   ;FOLD SPTP P710 CONT Vel=100 % PDAT71 Tool[1] Base[0] ;%{PE}
      ;FOLD Parameters ;%{h}
         ;Params IlfProvider=kukaroboter.basistech.inlineforms.movement.spline; Kuka.IsGlobalPoint=FALSE; Kuka.PointName=P710; Kuka.BlendingEnabled=TRUE; Kuka.MoveDataPtpName=PDAT71; Kuka.VelocityPtp=100; Kuka.VelocityFieldEnabled=TRUE; Kuka.ColDetectFieldEnabled=TRUE; Kuka.CurrentCDSetIndex=0; Kuka.MovementParameterFieldEnabled=TRUE; IlfCommand=SPTP
      ;ENDFOLD
      SPTP XP710 WITH $VEL_AXIS[1] = SVEL_JOINT(100.0), $TOOL = STOOL2(FP710), $BASE = SBASE(FP710.BASE_NO), $IPO_MODE = SIPO_MODE(FP710.IPO_FRAME), $LOAD = SLOAD(FP710.TOOL_NO), $ACC_AXIS[1] = SACC_JOINT(PPDAT71), $APO = SAPO_PTP(PPDAT71), $GEAR_JERK[1] = SGEAR_JERK(PPDAT71), $COLLMON_TOL_PRO[1] = USE_CM_PRO_VALUES(0) C_Spl
   ;ENDFOLD

   trigger when distance=0 delay=0 do B_Brenner_aktiv=FALSE
   trigger when distance=1 delay=0 do Brenner (I_n_aktive_Brenner,#loeschen) prio=-1
   ;FOLD SPTP P700 CONT Vel=100 % PDAT72 Tool[1] Base[0] ;%{PE}
      ;FOLD Parameters ;%{h}
         ;Params IlfProvider=kukaroboter.basistech.inlineforms.movement.spline; Kuka.IsGlobalPoint=FALSE; Kuka.PointName=P700; Kuka.BlendingEnabled=TRUE; Kuka.MoveDataPtpName=PDAT72; Kuka.VelocityPtp=100; Kuka.VelocityFieldEnabled=TRUE; Kuka.ColDetectFieldEnabled=TRUE; Kuka.CurrentCDSetIndex=0; Kuka.MovementParameterFieldEnabled=TRUE; IlfCommand=SPTP
      ;ENDFOLD
      SPTP XP700 WITH $VEL_AXIS[1] = SVEL_JOINT(100.0), $TOOL = STOOL2(FP700), $BASE = SBASE(FP700.BASE_NO), $IPO_MODE = SIPO_MODE(FP700.IPO_FRAME), $LOAD = SLOAD(FP700.TOOL_NO), $ACC_AXIS[1] = SACC_JOINT(PPDAT72), $APO = SAPO_PTP(PPDAT72), $GEAR_JERK[1] = SGEAR_JERK(PPDAT72), $COLLMON_TOL_PRO[1] = USE_CM_PRO_VALUES(0) C_Spl
   ;ENDFOLD

END

;***************************************************
;** Alternativprogramm ohne Bauteilbeflammen *******
;***************************************************

DEF ohne_Beflammen ()

   ;BEFLAMMEN WIRD NICHT VERWENDET
   RETURN

   ; hier Roboterbewegung

   trigger when distance=1 delay=0 do UmgreifStation_Pos (#auf) prio=-1
   ;FOLD SPTP P1000 CONT Vel=100 % PDAT73 Tool[1] Base[0] ;%{PE}
      ;FOLD Parameters ;%{h}
         ;Params IlfProvider=kukaroboter.basistech.inlineforms.movement.spline; Kuka.IsGlobalPoint=FALSE; Kuka.PointName=P1000; Kuka.BlendingEnabled=TRUE; Kuka.MoveDataPtpName=PDAT73; Kuka.VelocityPtp=100; Kuka.VelocityFieldEnabled=TRUE; Kuka.ColDetectFieldEnabled=TRUE; Kuka.CurrentCDSetIndex=0; Kuka.MovementParameterFieldEnabled=TRUE; IlfCommand=SPTP
      ;ENDFOLD
      SPTP XP1000 WITH $VEL_AXIS[1] = SVEL_JOINT(100.0), $TOOL = STOOL2(FP1000), $BASE = SBASE(FP1000.BASE_NO), $IPO_MODE = SIPO_MODE(FP1000.IPO_FRAME), $LOAD = SLOAD(FP1000.TOOL_NO), $ACC_AXIS[1] = SACC_JOINT(PPDAT73), $APO = SAPO_PTP(PPDAT73), $GEAR_JERK[1] = SGEAR_JERK(PPDAT73), $COLLMON_TOL_PRO[1] = USE_CM_PRO_VALUES(0) C_Spl
   ;ENDFOLD

   continue
   if ((E_mit_Bedrucken==TRUE) and (B_Ausschuss==FALSE)) then ; $IN[1201] mit Bedrucken von SPS
      trigger when distance=1 delay=0 do drucker(#druck)prio=-1

   endif ; and (E_WAAGE_TEIL_IO)

   ;FOLD SPTP P1010 CONT Vel=100 % PDAT74 Tool[1] Base[0] ;%{PE}
      ;FOLD Parameters ;%{h}
         ;Params IlfProvider=kukaroboter.basistech.inlineforms.movement.spline; Kuka.IsGlobalPoint=FALSE; Kuka.PointName=P1010; Kuka.BlendingEnabled=TRUE; Kuka.MoveDataPtpName=PDAT74; Kuka.VelocityPtp=100; Kuka.VelocityFieldEnabled=TRUE; Kuka.ColDetectFieldEnabled=TRUE; Kuka.CurrentCDSetIndex=0; Kuka.MovementParameterFieldEnabled=TRUE; IlfCommand=SPTP
      ;ENDFOLD
      SPTP XP1010 WITH $VEL_AXIS[1] = SVEL_JOINT(100.0), $TOOL = STOOL2(FP1010), $BASE = SBASE(FP1010.BASE_NO), $IPO_MODE = SIPO_MODE(FP1010.IPO_FRAME), $LOAD = SLOAD(FP1010.TOOL_NO), $ACC_AXIS[1] = SACC_JOINT(PPDAT74), $APO = SAPO_PTP(PPDAT74), $GEAR_JERK[1] = SGEAR_JERK(PPDAT74), $COLLMON_TOL_PRO[1] = USE_CM_PRO_VALUES(0) C_Spl
   ;ENDFOLD

   if ((E_mit_Bedrucken==TRUE) and (B_Ausschuss==FALSE)) then ; $IN[1201] mit Bedrucken von SPS
      ; and (E_WAAGE_TEIL_IO)

      ;FOLD SPTP P1020 CONT Vel=100 % PDAT75 Tool[1] Base[0] ;%{PE}
         ;FOLD Parameters ;%{h}
            ;Params IlfProvider=kukaroboter.basistech.inlineforms.movement.spline; Kuka.IsGlobalPoint=FALSE; Kuka.PointName=P1020; Kuka.BlendingEnabled=TRUE; Kuka.MoveDataPtpName=PDAT75; Kuka.VelocityPtp=100; Kuka.VelocityFieldEnabled=TRUE; Kuka.ColDetectFieldEnabled=TRUE; Kuka.CurrentCDSetIndex=0; Kuka.MovementParameterFieldEnabled=TRUE; IlfCommand=SPTP
         ;ENDFOLD
         SPTP XP1020 WITH $VEL_AXIS[1] = SVEL_JOINT(100.0), $TOOL = STOOL2(FP1020), $BASE = SBASE(FP1020.BASE_NO), $IPO_MODE = SIPO_MODE(FP1020.IPO_FRAME), $LOAD = SLOAD(FP1020.TOOL_NO), $ACC_AXIS[1] = SACC_JOINT(PPDAT75), $APO = SAPO_PTP(PPDAT75), $GEAR_JERK[1] = SGEAR_JERK(PPDAT75), $COLLMON_TOL_PRO[1] = USE_CM_PRO_VALUES(0) C_Spl
      ;ENDFOLD
   endif

end
;***************************************************
;** Alternativprogramm ohne Bauteil bedrucken ******
;***************************************************

DEF ohne_RFID()

   ;Umorientierung wenn ohne RFID produziert wird

   ;FOLD SPTP P2000 CONT Vel=100 % PDAT76 Tool[1] Base[0] ;%{PE}
      ;FOLD Parameters ;%{h}
         ;Params IlfProvider=kukaroboter.basistech.inlineforms.movement.spline; Kuka.IsGlobalPoint=FALSE; Kuka.PointName=P2000; Kuka.BlendingEnabled=TRUE; Kuka.MoveDataPtpName=PDAT76; Kuka.VelocityPtp=100; Kuka.VelocityFieldEnabled=TRUE; Kuka.ColDetectFieldEnabled=TRUE; Kuka.CurrentCDSetIndex=0; Kuka.MovementParameterFieldEnabled=TRUE; IlfCommand=SPTP
      ;ENDFOLD
      SPTP XP2000 WITH $VEL_AXIS[1] = SVEL_JOINT(100.0), $TOOL = STOOL2(FP2000), $BASE = SBASE(FP2000.BASE_NO), $IPO_MODE = SIPO_MODE(FP2000.IPO_FRAME), $LOAD = SLOAD(FP2000.TOOL_NO), $ACC_AXIS[1] = SACC_JOINT(PPDAT76), $APO = SAPO_PTP(PPDAT76), $GEAR_JERK[1] = SGEAR_JERK(PPDAT76), $COLLMON_TOL_PRO[1] = USE_CM_PRO_VALUES(0) C_Spl
   ;ENDFOLD

   ;FOLD SPTP P2010 CONT Vel=100 % PDAT77 Tool[1] Base[0] ;%{PE}
      ;FOLD Parameters ;%{h}
         ;Params IlfProvider=kukaroboter.basistech.inlineforms.movement.spline; Kuka.IsGlobalPoint=FALSE; Kuka.PointName=P2010; Kuka.BlendingEnabled=TRUE; Kuka.MoveDataPtpName=PDAT77; Kuka.VelocityPtp=100; Kuka.VelocityFieldEnabled=TRUE; Kuka.ColDetectFieldEnabled=TRUE; Kuka.CurrentCDSetIndex=0; Kuka.MovementParameterFieldEnabled=TRUE; IlfCommand=SPTP
      ;ENDFOLD
      SPTP XP2010 WITH $VEL_AXIS[1] = SVEL_JOINT(100.0), $TOOL = STOOL2(FP2010), $BASE = SBASE(FP2010.BASE_NO), $IPO_MODE = SIPO_MODE(FP2010.IPO_FRAME), $LOAD = SLOAD(FP2010.TOOL_NO), $ACC_AXIS[1] = SACC_JOINT(PPDAT77), $APO = SAPO_PTP(PPDAT77), $GEAR_JERK[1] = SGEAR_JERK(PPDAT77), $COLLMON_TOL_PRO[1] = USE_CM_PRO_VALUES(0) C_Spl
   ;ENDFOLD

   ;FOLD SPTP P2020 CONT Vel=100 % PDAT78 Tool[1] Base[0] ;%{PE}
      ;FOLD Parameters ;%{h}
         ;Params IlfProvider=kukaroboter.basistech.inlineforms.movement.spline; Kuka.IsGlobalPoint=FALSE; Kuka.PointName=P2020; Kuka.BlendingEnabled=TRUE; Kuka.MoveDataPtpName=PDAT78; Kuka.VelocityPtp=100; Kuka.VelocityFieldEnabled=TRUE; Kuka.ColDetectFieldEnabled=TRUE; Kuka.CurrentCDSetIndex=0; Kuka.MovementParameterFieldEnabled=TRUE; IlfCommand=SPTP
      ;ENDFOLD
      SPTP XP2020 WITH $VEL_AXIS[1] = SVEL_JOINT(100.0), $TOOL = STOOL2(FP2020), $BASE = SBASE(FP2020.BASE_NO), $IPO_MODE = SIPO_MODE(FP2020.IPO_FRAME), $LOAD = SLOAD(FP2020.TOOL_NO), $ACC_AXIS[1] = SACC_JOINT(PPDAT78), $APO = SAPO_PTP(PPDAT78), $GEAR_JERK[1] = SGEAR_JERK(PPDAT78), $COLLMON_TOL_PRO[1] = USE_CM_PRO_VALUES(0) C_Spl
   ;ENDFOLD

end

;***************************************************
;** Programm, um rueckwaerts aus der Form bis vor **
;***        Teileaufnahme zu fahren              ***
;***************************************************

DEF  RRaus ( )

   INT i

   B_Ausschuss=TRUE
   $ov_pro=10
   BAS (#vel_cp,1.0)
   BAS (#vel_ptp,50)

   ventile_aus ()

   $BASE=Base_Data[1]
   $TOOL=Tool_Data[1]

   wait for (E_SGM_Form_auf==TRUE) ; $IN[3] SGM Form offen (E67)
   if ($flag[7]==TRUE) then
      LIN  XP100
   endif

   if ($flag[6]==TRUE) then
      LIN  XP40
   endif

   if ($flag[5]==TRUE) then
      LIN  XP35
   endif

   if ($flag[4]==TRUE) then
      LIN  XP30
   endif

   if ($flag[3]==TRUE) then
      PTP XP20
   endif

   if ($flag[2]==TRUE) then
      PTP XP10
   endif

   if ($flag[1]==TRUE) then
      PTP XHome
   else
      Meldung (#notify,10)
      Meldung (#quit,27)
      loop
         HALT  ;Roboter von Hand aus der Form fahren !!!
      endloop
   endif

   for i=1 to 10
      $flag[i]=FALSE
   endfor

   B_GST_war_gedrueckt=FALSE
   ;B_L_Start=FALSE
   B_Teilaufnahme=TRUE

END

;***************************************************
;** Programm, zum Uberpruefen der Endlagen der   **
;***            Benutzerventile                  ***
;***************************************************

Def Chk_BV (BV_Nr: in,BV_Zustand: in)

   INT BV_Nr
   DECL Mode2 BV_Zustand

   ;fold  Greiferbelegung, Stand: 02.11.2020
      ;***************************************************
      ;  V1  = Teilevakuum vorne
      ;  V2  = n.v.
      ;  V3  = Teilevakuum vorne unten ;nur ab Umgreifstation
      ;  V4  = Teilevakuum hinten unten ;nur ab Umgreifstation
      ;  BV1/AS = Teilegreifer schließen
      ;  BV1/GS = n.v.
      ;  BV2/AS = Teilegreifer hinten langer hub nach vorne
      ;  BV2/GS = Teilegreifer hinten langer hub nach hinten
      ;  BV3/AS = Teilegreifer hinten kurzer hub nach vorne
      ;  BV3/GS = Teilegreifer hinten kurzer hub nach hinten
      ;  BV4/AS = Angussgreifer schließen
      ;  BV4/GS = n.v.
      ;  BV5/AS = Angussschneider nach vorne
      ;  BV5/GS = Angussschneider nach hinten
      ;  BV6/AS = Angussschneider schließen
      ;***************************************************
   ;endfold

   switch BV_Nr

      ; Benutzerventil 1 = Teilegreifer
      case 1

         switch BV_Zustand

            case #GS

            case #AS

               wait for (E_ASi_22_3==TRUE); IN 363(Abf. Radl oben links)
               wait for (E_ASi_22_4==TRUE); IN 364(Abf. Dreilaendereck links)
               wait for (E_ASi_24_3==TRUE); IN 379(Abf. Radl unten links)
               wait for (E_ASi_26_3==TRUE); IN 395(Abf. Radl oben rechts)
               wait for (E_ASi_26_4==TRUE); IN 496(Abf. Dreilaendereck rechts)
               wait for (E_ASi_28_3==TRUE); IN 411(Abf. Radlauf unten rechts)

         endswitch

         ; Benutzerventil 2 =  Teilegreifer hinten langer hub
      case 2

         switch BV_Zustand

            case #GS

               wait for (E_ASi_22_1==TRUE)
               wait for (E_ASi_24_1==TRUE)
               wait for (E_ASi_26_1==TRUE)
               wait for (E_ASi_28_1==TRUE)

            case #AS

               wait for (E_ASi_22_2==TRUE)
               wait for (E_ASi_24_2==TRUE)
               wait for (E_ASi_26_2==TRUE)
               wait for (E_ASi_28_2==TRUE)

         endswitch

         ; Benutzerventil 3 = none
      case 3

         switch BV_Zustand

            case #GS

            case #AS

         endswitch

         ; Benutzerventil 4 = Angussgreifer
      case 4

         switch BV_Zustand

            case #GS

            case #AS

               wait for (E_ASi_23_1==TRUE); IN 369(Anguss links)
               wait for (E_ASi_23_2==TRUE); IN 370(Anguss rechts)
               wait for (E_ASi_27_1==TRUE); IN 401(Anguss rechts)

         endswitch

         ; Benutzerventil 5 = none
      case 5

         switch BV_Zustand

            case #GS

            case #AS

         endswitch

         ; Benutzerventil 6 = none
      case 6

         switch BV_Zustand

            case #GS

            case #AS

         endswitch

      default
         loop
            halt ; BV nicht vorhanden
         endloop

   endswitch

end

;***************************************************
;*** Teileabfrage Vakuumkreise und ASI Eingänge  ***
;***************************************************

DEF Teileabfrage()

   wait for (E_VK1==TRUE)
   ;wait for (E_VK2==TRUE)
   ;wait for (E_VK3==TRUE)
   ;wait for (E_VK4==TRUE)
   wait for (E_ASi_22_3==TRUE); IN 363(Abf. Radl oben links)
   wait for (E_ASi_22_4==TRUE); IN 364(Abf. Dreilaendereck links)
   wait for (E_ASi_23_1==TRUE); IN 369(Anguss links)
   wait for (E_ASi_23_2==TRUE); IN 370(Anguss rechts)
   wait for (E_ASi_24_3==TRUE); IN 379(Abf. Radl unten links)
   wait for (E_ASi_26_3==TRUE); IN 395(Abf. Radl oben rechts)
   wait for (E_ASi_26_4==TRUE); IN 496(Abf. Dreilaendereck rechts)
   wait for (E_ASi_27_1==TRUE); IN 401(Anguss rechts)
   wait for (E_ASi_28_3==TRUE); IN 411(Abf. Radlauf unten rechts)

End

--- sp15_005.dat ---
&ACCESS RVO1
&REL 244
&PARAM DISKPATH = KRC:\R1\Program\Bauteilprogramme
DEFDAT  SP15_005
;FOLD EXTERNAL DECLARATIONS;%{PE}%MKUKATPBASIS,%CEXT,%VCOMMON,%P
;FOLD BASISTECH EXT;%{PE}%MKUKATPBASIS,%CEXT,%VEXT,%P
EXT  BAS (BAS_COMMAND  :IN,REAL  :IN )
;ENDFOLD (BASISTECH EXT)
;FOLD USER EXT;%{E}%MKUKATPUSER,%CEXT,%VEXT,%P
;Make your modifications here

;ENDFOLD (USER EXT)
;ENDFOLD (EXTERNAL DECLARATIONS)

;***************************************************
;Common Declarations********************************
;***************************************************
DECL E6POS XP200={X 2198.25366,Y -125.542969,Z 1747.09790,A 176.729721,B 44.9991875,C 179.999023,S 2,T 34,E1 0.0,E2 0.0,E3 0.0,E4 0.0,E5 0.0,E6 0.0}
DECL FDAT FP200={TOOL_NO 1,BASE_NO 0,IPO_FRAME #BASE,POINT2[] " "}
DECL PDAT PPDAT6={VEL 100.000,ACC 100.000,APO_DIST 500.000,APO_MODE #CDIS,GEAR_JERK 100.000,EXAX_IGN 0}


;***************************************************
;SGM Declarations***********************************
;***************************************************
DECL E6POS XP10={X 1853.22363,Y 1615.74561,Z 1754.75720,A 60.7845039,B -43.4993439,C -175.197784,S 2,T 43,E1 0.0,E2 0.0,E3 0.0,E4 0.0,E5 0.0,E6 0.0}
DECL FDAT FP10={TOOL_NO 1,BASE_NO 0,IPO_FRAME #BASE,POINT2[] " "}
DECL PDAT PPDAT1={VEL 100.000,ACC 100.000,APO_DIST 250.000,APO_MODE #CDIS,GEAR_JERK 100.000,EXAX_IGN 0}

DECL E6POS XP20={X 1174.55273,Y 2717.27319,Z 949.700256,A -0.590916,B 44.9981651,C 179.820206,S 2,T 43,E1 0.0,E2 0.0,E3 0.0,E4 0.0,E5 0.0,E6 0.0}
DECL FDAT FP20={TOOL_NO 1,BASE_NO 0,IPO_FRAME #BASE,POINT2[] " "}
DECL PDAT PPDAT2={VEL 100.000,ACC 100.000,APO_DIST 250.000,APO_MODE #CDIS,GEAR_JERK 100.000,EXAX_IGN 0}

DECL E6POS XP30={X 1174.55273,Y 2717.27319,Z 118.860199,A -0.590916097,B 44.9981651,C 179.820206,S 2,T 43,E1 0.0,E2 0.0,E3 0.0,E4 0.0,E5 0.0,E6 0.0}
DECL FDAT FP30={TOOL_NO 1,BASE_NO 0,IPO_FRAME #BASE,POINT2[] " "}
DECL PDAT PPDAT3={VEL 100.000,ACC 100.000,APO_DIST 250.000,APO_MODE #CDIS,GEAR_JERK 100.000,EXAX_IGN 0}

DECL E6POS XP35={X 1174.55273,Y 2717.27319,Z -593.502808,A -0.590916157,B 44.9981651,C 179.820206,S 2,T 43,E1 0.0,E2 0.0,E3 0.0,E4 0.0,E5 0.0,E6 0.0}
DECL FDAT FP35={TOOL_NO 1,BASE_NO 0,IPO_FRAME #BASE,POINT2[] " "}
DECL LDAT LCPDAT1={VEL 2.00000,ACC 100.000,APO_DIST 250.000,APO_FAC 50.0000,AXIS_VEL 100.000,AXIS_ACC 100.000,ORI_TYP #VAR,CIRC_TYP #BASE,JERK_FAC 50.0000,GEAR_JERK 100.000,EXAX_IGN 0,CB {AUX_PT {ORI #CONSIDER,E1 #CONSIDER,E2 #CONSIDER,E3 #CONSIDER,E4 #CONSIDER,E5 #CONSIDER,E6 #CONSIDER},TARGET_PT {ORI #INTERPOLATE,E1 #INTERPOLATE,E2 #INTERPOLATE,E3 #INTERPOLATE,E4 #INTERPOLATE,E5 #INTERPOLATE,E6 #INTERPOLATE}}}

DECL E6POS XP40={X 1174.55273,Y 2717.27319,Z -1291.60657,A -0.590916276,B 44.9981651,C 179.820206,S 2,T 41,E1 0.0,E2 0.0,E3 0.0,E4 0.0,E5 0.0,E6 0.0}
DECL FDAT FP40={TOOL_NO 1,BASE_NO 0,IPO_FRAME #BASE,POINT2[] " "}
DECL LDAT LCPDAT2={VEL 2.00000,ACC 100.000,APO_DIST 150.000,APO_FAC 50.0000,AXIS_VEL 100.000,AXIS_ACC 100.000,ORI_TYP #VAR,CIRC_TYP #BASE,JERK_FAC 50.0000,GEAR_JERK 100.000,EXAX_IGN 0,CB {AUX_PT {ORI #CONSIDER,E1 #CONSIDER,E2 #CONSIDER,E3 #CONSIDER,E4 #CONSIDER,E5 #CONSIDER,E6 #CONSIDER},TARGET_PT {ORI #INTERPOLATE,E1 #INTERPOLATE,E2 #INTERPOLATE,E3 #INTERPOLATE,E4 #INTERPOLATE,E5 #INTERPOLATE,E6 #INTERPOLATE}}}

DECL E6POS XP100={X 589.207214,Y 2717.27319,Z -1291.60657,A -0.590916336,B 44.9981651,C 179.820206,S 2,T 41,E1 0.0,E2 0.0,E3 0.0,E4 0.0,E5 0.0,E6 0.0}
DECL FDAT FP100={TOOL_NO 1,BASE_NO 0,IPO_FRAME #BASE,POINT2[] " "}
DECL LDAT LCPDAT3={VEL 1.00000,ACC 100.000,APO_DIST 250.000,APO_FAC 50.0000,AXIS_VEL 100.000,AXIS_ACC 100.000,ORI_TYP #VAR,CIRC_TYP #BASE,JERK_FAC 50.0000,GEAR_JERK 100.000,EXAX_IGN 0,CB {AUX_PT {ORI #CONSIDER,E1 #CONSIDER,E2 #CONSIDER,E3 #CONSIDER,E4 #CONSIDER,E5 #CONSIDER,E6 #CONSIDER},TARGET_PT {ORI #INTERPOLATE,E1 #INTERPOLATE,E2 #INTERPOLATE,E3 #INTERPOLATE,E4 #INTERPOLATE,E5 #INTERPOLATE,E6 #INTERPOLATE}}}
DECL LDAT LCPDAT4={VEL 1.00000,ACC 100.000,APO_DIST 250.000,APO_FAC 50.0000,AXIS_VEL 100.000,AXIS_ACC 100.000,ORI_TYP #VAR,CIRC_TYP #BASE,JERK_FAC 50.0000,GEAR_JERK 100.000,EXAX_IGN 0,CB {AUX_PT {ORI #CONSIDER,E1 #CONSIDER,E2 #CONSIDER,E3 #CONSIDER,E4 #CONSIDER,E5 #CONSIDER,E6 #CONSIDER},TARGET_PT {ORI #INTERPOLATE,E1 #INTERPOLATE,E2 #INTERPOLATE,E3 #INTERPOLATE,E4 #INTERPOLATE,E5 #INTERPOLATE,E6 #INTERPOLATE}}}

DECL E6POS XP102={X 625.272339,Y 2717.27319,Z -1291.60657,A -0.590916336,B 44.9981651,C 179.820206,S 2,T 41,E1 0.0,E2 0.0,E3 0.0,E4 0.0,E5 0.0,E6 0.0}
DECL FDAT FP102={TOOL_NO 1,BASE_NO 0,IPO_FRAME #BASE,POINT2[] " "}
DECL LDAT LCPDAT5={VEL 1.00000,ACC 100.000,APO_DIST 250.000,APO_FAC 50.0000,AXIS_VEL 100.000,AXIS_ACC 100.000,ORI_TYP #VAR,CIRC_TYP #BASE,JERK_FAC 50.0000,GEAR_JERK 100.000,EXAX_IGN 0,CB {AUX_PT {ORI #CONSIDER,E1 #CONSIDER,E2 #CONSIDER,E3 #CONSIDER,E4 #CONSIDER,E5 #CONSIDER,E6 #CONSIDER},TARGET_PT {ORI #INTERPOLATE,E1 #INTERPOLATE,E2 #INTERPOLATE,E3 #INTERPOLATE,E4 #INTERPOLATE,E5 #INTERPOLATE,E6 #INTERPOLATE}}}
DECL LDAT LCPDAT6={VEL 2.00000,ACC 100.000,APO_DIST 400.000,APO_FAC 50.0000,AXIS_VEL 100.000,AXIS_ACC 100.000,ORI_TYP #VAR,CIRC_TYP #BASE,JERK_FAC 50.0000,GEAR_JERK 100.000,EXAX_IGN 0,CB {AUX_PT {ORI #CONSIDER,E1 #CONSIDER,E2 #CONSIDER,E3 #CONSIDER,E4 #CONSIDER,E5 #CONSIDER,E6 #CONSIDER},TARGET_PT {ORI #INTERPOLATE,E1 #INTERPOLATE,E2 #INTERPOLATE,E3 #INTERPOLATE,E4 #INTERPOLATE,E5 #INTERPOLATE,E6 #INTERPOLATE}}}
DECL LDAT LCPDAT7={VEL 2.00000,ACC 100.000,APO_DIST 250.000,APO_FAC 50.0000,AXIS_VEL 100.000,AXIS_ACC 100.000,ORI_TYP #VAR,CIRC_TYP #BASE,JERK_FAC 50.0000,GEAR_JERK 100.000,EXAX_IGN 0,CB {AUX_PT {ORI #CONSIDER,E1 #CONSIDER,E2 #CONSIDER,E3 #CONSIDER,E4 #CONSIDER,E5 #CONSIDER,E6 #CONSIDER},TARGET_PT {ORI #INTERPOLATE,E1 #INTERPOLATE,E2 #INTERPOLATE,E3 #INTERPOLATE,E4 #INTERPOLATE,E5 #INTERPOLATE,E6 #INTERPOLATE}}}
DECL LDAT LCPDAT8={VEL 2.00000,ACC 100.000,APO_DIST 250.000,APO_FAC 50.0000,AXIS_VEL 100.000,AXIS_ACC 100.000,ORI_TYP #VAR,CIRC_TYP #BASE,JERK_FAC 50.0000,GEAR_JERK 100.000,EXAX_IGN 0,CB {AUX_PT {ORI #CONSIDER,E1 #CONSIDER,E2 #CONSIDER,E3 #CONSIDER,E4 #CONSIDER,E5 #CONSIDER,E6 #CONSIDER},TARGET_PT {ORI #INTERPOLATE,E1 #INTERPOLATE,E2 #INTERPOLATE,E3 #INTERPOLATE,E4 #INTERPOLATE,E5 #INTERPOLATE,E6 #INTERPOLATE}}}
DECL PDAT PPDAT4={VEL 100.000,ACC 100.000,APO_DIST 500.000,APO_MODE #CDIS,GEAR_JERK 100.000,EXAX_IGN 0}
DECL PDAT PPDAT5={VEL 100.000,ACC 100.000,APO_DIST 500.000,APO_MODE #CDIS,GEAR_JERK 100.000,EXAX_IGN 0}

;***************************************************
;Conveyour Declarations*****************************
;***************************************************
;common positions for both conveyours
DECL E6POS XP1900={X 1008.73590,Y -1708.91467,Z 1056.99243,A -31.9333897,B 52.9364738,C 16.7323208,S 2,T 10,E1 0.0,E2 0.0,E3 0.0,E4 0.0,E5 0.0,E6 0.0}
DECL FDAT FP1900={TOOL_NO 1,BASE_NO 0,IPO_FRAME #BASE,POINT2[] " "}
DECL PDAT PPDAT7={VEL 100.000,ACC 100.000,APO_DIST 250.000,APO_MODE #CDIS,GEAR_JERK 100.000,EXAX_IGN 0}
DECL E6POS XP1910={X 616.562927,Y -2628.79199,Z -65.0746231,A 1.20445049,B 66.1203766,C 87.5318527,S 2,T 10,E1 0.0,E2 0.0,E3 0.0,E4 0.0,E5 0.0,E6 0.0}
DECL FDAT FP1910={TOOL_NO 1,BASE_NO 0,IPO_FRAME #BASE,POINT2[] " "}
DECL PDAT PPDAT8={VEL 100.000,ACC 100.000,APO_DIST 250.000,APO_MODE #CDIS,GEAR_JERK 100.000,EXAX_IGN 0}
DECL E6POS XP1920={X -390.418793,Y -2601.90039,Z -699.180176,A 45.1227570,B 59.2144775,C -164.045944,S 2,T 10,E1 0.0,E2 0.0,E3 0.0,E4 0.0,E5 0.0,E6 0.0}
DECL FDAT FP1920={TOOL_NO 1,BASE_NO 0,IPO_FRAME #BASE,POINT2[] " "}
DECL PDAT PPDAT9={VEL 100.000,ACC 100.000,APO_DIST 250.000,APO_MODE #CDIS,GEAR_JERK 100.000,EXAX_IGN 0}

;conveyour 1 unten
DECL E6POS XP1930_unten={X 1013.42212,Y -2233.39673,Z -865.971130,A -0.708070934,B 42.4057236,C 179.320618,S 2,T 10,E1 0.0,E2 0.0,E3 0.0,E4 0.0,E5 0.0,E6 0.0}
DECL FDAT FP1930_unten={TOOL_NO 1,BASE_NO 0,IPO_FRAME #BASE,POINT2[] " "}

DECL E6POS XP1940_unten={X -401.907135,Y -2154.10303,Z -857.722778,A -0.0218503568,B 36.5302429,C 179.871857,S 2,T 10,E1 0.0,E2 0.0,E3 0.0,E4 0.0,E5 0.0,E6 0.0}
DECL FDAT FP1940_unten={TOOL_NO 1,BASE_NO 0,IPO_FRAME #BASE,POINT2[] " "}
DECL PDAT PPDAT21={VEL 100.000,ACC 100.000,APO_DIST 350.000,APO_MODE #CDIS,GEAR_JERK 100.000,EXAX_IGN 0}

DECL E6POS XP1950_unten={X -401.907135,Y -2154.10303,Z -1529.26611,A -0.0218503587,B 36.5302429,C 179.871857,S 2,T 8,E1 0.0,E2 0.0,E3 0.0,E4 0.0,E5 0.0,E6 0.0}
DECL FDAT FP1950_unten={TOOL_NO 1,BASE_NO 0,IPO_FRAME #BASE,POINT2[] " "}
DECL LDAT LCPDAT11={VEL 1.00000,ACC 100.000,APO_DIST 500.000,APO_FAC 50.0000,AXIS_VEL 100.000,AXIS_ACC 100.000,ORI_TYP #VAR,CIRC_TYP #BASE,JERK_FAC 50.0000,GEAR_JERK 100.000,EXAX_IGN 0,CB {AUX_PT {ORI #CONSIDER,E1 #CONSIDER,E2 #CONSIDER,E3 #CONSIDER,E4 #CONSIDER,E5 #CONSIDER,E6 #CONSIDER},TARGET_PT {ORI #INTERPOLATE,E1 #INTERPOLATE,E2 #INTERPOLATE,E3 #INTERPOLATE,E4 #INTERPOLATE,E5 #INTERPOLATE,E6 #INTERPOLATE}}}
DECL LDAT LCPDAT12={VEL 1.00000,ACC 100.000,APO_DIST 350.000,APO_FAC 50.0000,AXIS_VEL 100.000,AXIS_ACC 100.000,ORI_TYP #VAR,CIRC_TYP #BASE,JERK_FAC 50.0000,GEAR_JERK 100.000,EXAX_IGN 0,CB {AUX_PT {ORI #CONSIDER,E1 #CONSIDER,E2 #CONSIDER,E3 #CONSIDER,E4 #CONSIDER,E5 #CONSIDER,E6 #CONSIDER},TARGET_PT {ORI #INTERPOLATE,E1 #INTERPOLATE,E2 #INTERPOLATE,E3 #INTERPOLATE,E4 #INTERPOLATE,E5 #INTERPOLATE,E6 #INTERPOLATE}}}
DECL PDAT PPDAT22={VEL 100.000,ACC 100.000,APO_DIST 350.000,APO_MODE #CDIS,GEAR_JERK 100.000,EXAX_IGN 0}
DECL PDAT PPDAT23={VEL 100.000,ACC 100.000,APO_DIST 500.000,APO_MODE #CDIS,GEAR_JERK 100.000,EXAX_IGN 0}
DECL PDAT PPDAT24={VEL 100.000,ACC 100.000,APO_DIST 500.000,APO_MODE #CDIS,GEAR_JERK 100.000,EXAX_IGN 0}
DECL PDAT PPDAT25={VEL 100.000,ACC 100.000,APO_DIST 500.000,APO_MODE #CDIS,GEAR_JERK 100.000,EXAX_IGN 0}
DECL PDAT PPDAT26={VEL 100.000,ACC 100.000,APO_DIST 500.000,APO_MODE #CDIS,GEAR_JERK 100.000,EXAX_IGN 0}


;conveyour 1 oben
DECL E6POS XP1930={X 2286.18115,Y 0.000230411548,Z 1849.57446,A -179.999893,B 66.9998779,C -179.999878,S 2,T 35,E1 0.0,E2 0.0,E3 0.0,E4 0.0,E5 0.0,E6 0.0}
DECL FDAT FP1930={TOOL_NO 1,BASE_NO 0,IPO_FRAME #BASE,POINT2[] " "}
DECL PDAT PPDAT10={VEL 100.000,ACC 100.000,APO_DIST 250.000,APO_MODE #CDIS,GEAR_JERK 100.000,EXAX_IGN 0}

DECL E6POS XP1940={X 2286.18115,Y 0.000230411548,Z 1849.57446,A -179.999893,B 66.9998779,C -179.999878,S 2,T 35,E1 0.0,E2 0.0,E3 0.0,E4 0.0,E5 0.0,E6 0.0}
DECL FDAT FP1940={TOOL_NO 1,BASE_NO 0,IPO_FRAME #BASE,POINT2[] " "}
DECL PDAT PPDAT11={VEL 100.000,ACC 100.000,APO_DIST 250.000,APO_MODE #CDIS,GEAR_JERK 100.000,EXAX_IGN 0}

DECL E6POS XP1950={X 2286.18115,Y 0.000230411548,Z 1849.57446,A -179.999893,B 66.9998779,C -179.999878,S 2,T 35,E1 0.0,E2 0.0,E3 0.0,E4 0.0,E5 0.0,E6 0.0}
DECL FDAT FP1950={TOOL_NO 1,BASE_NO 0,IPO_FRAME #BASE,POINT2[] " "}
DECL LDAT LCPDAT9={VEL 0.500000,ACC 100.000,APO_DIST 500.000,APO_FAC 50.0000,AXIS_VEL 100.000,AXIS_ACC 100.000,ORI_TYP #VAR,CIRC_TYP #BASE,JERK_FAC 50.0000,GEAR_JERK 100.000,EXAX_IGN 0,CB {AUX_PT {ORI #CONSIDER,E1 #CONSIDER,E2 #CONSIDER,E3 #CONSIDER,E4 #CONSIDER,E5 #CONSIDER,E6 #CONSIDER},TARGET_PT {ORI #INTERPOLATE,E1 #INTERPOLATE,E2 #INTERPOLATE,E3 #INTERPOLATE,E4 #INTERPOLATE,E5 #INTERPOLATE,E6 #INTERPOLATE}}}
DECL LDAT LCPDAT10={VEL 0.500000,ACC 100.000,APO_DIST 500.000,APO_FAC 50.0000,AXIS_VEL 100.000,AXIS_ACC 100.000,ORI_TYP #VAR,CIRC_TYP #BASE,JERK_FAC 50.0000,GEAR_JERK 100.000,EXAX_IGN 0,CB {AUX_PT {ORI #CONSIDER,E1 #CONSIDER,E2 #CONSIDER,E3 #CONSIDER,E4 #CONSIDER,E5 #CONSIDER,E6 #CONSIDER},TARGET_PT {ORI #INTERPOLATE,E1 #INTERPOLATE,E2 #INTERPOLATE,E3 #INTERPOLATE,E4 #INTERPOLATE,E5 #INTERPOLATE,E6 #INTERPOLATE}}}
DECL PDAT PPDAT13={VEL 100.000,ACC 100.000,APO_DIST 250.000,APO_MODE #CDIS,GEAR_JERK 100.000,EXAX_IGN 0}
DECL PDAT PPDAT14={VEL 100.000,ACC 100.000,APO_DIST 250.000,APO_MODE #CDIS,GEAR_JERK 100.000,EXAX_IGN 0}
DECL PDAT PPDAT15={VEL 100.000,ACC 100.000,APO_DIST 250.000,APO_MODE #CDIS,GEAR_JERK 100.000,EXAX_IGN 0}
DECL PDAT PPDAT16={VEL 100.000,ACC 100.000,APO_DIST 250.000,APO_MODE #CDIS,GEAR_JERK 100.000,EXAX_IGN 0}
DECL PDAT PPDAT17={VEL 100.000,ACC 100.000,APO_DIST 250.000,APO_MODE #CDIS,GEAR_JERK 100.000,EXAX_IGN 0}
DECL PDAT PPDAT18={VEL 100.000,ACC 100.000,APO_DIST 500.000,APO_MODE #CDIS,GEAR_JERK 100.000,EXAX_IGN 0}
DECL PDAT PPDAT19={VEL 100.000,ACC 100.000,APO_DIST 250.000,APO_MODE #CDIS,GEAR_JERK 100.000,EXAX_IGN 0}
DECL PDAT PPDAT20={VEL 100.000,ACC 100.000,APO_DIST 350.000,APO_MODE #CDIS,GEAR_JERK 100.000,EXAX_IGN 0}

;***************************************************
;Sprue Cutter Declarations**************************
;***************************************************
DECL E6POS XP300={X 2286.18115,Y 0.000230411548,Z 1849.57446,A -179.999893,B 66.9998779,C -179.999878,S 2,T 35,E1 0.0,E2 0.0,E3 0.0,E4 0.0,E5 0.0,E6 0.0}
DECL FDAT FP300={TOOL_NO 1,BASE_NO 0,IPO_FRAME #BASE,POINT2[] " "}
DECL PDAT PPDAT27={VEL 50.0000,ACC 100.000,APO_DIST 250.000,APO_MODE #CDIS,GEAR_JERK 100.000,EXAX_IGN 0}

DECL E6POS XP310={X 2286.18115,Y 0.000230411548,Z 1849.57446,A -179.999893,B 66.9998779,C -179.999878,S 2,T 35,E1 0.0,E2 0.0,E3 0.0,E4 0.0,E5 0.0,E6 0.0}
DECL FDAT FP310={TOOL_NO 1,BASE_NO 0,IPO_FRAME #BASE,POINT2[] " "}
DECL PDAT PPDAT28={VEL 50.0000,ACC 100.000,APO_DIST 250.000,APO_MODE #CDIS,GEAR_JERK 100.000,EXAX_IGN 0}

DECL E6POS XP320={X 2286.18115,Y 0.000230411548,Z 1849.57446,A -179.999893,B 66.9998779,C -179.999878,S 2,T 35,E1 0.0,E2 0.0,E3 0.0,E4 0.0,E5 0.0,E6 0.0}
DECL FDAT FP320={TOOL_NO 1,BASE_NO 0,IPO_FRAME #BASE,POINT2[] " "}
DECL PDAT PPDAT29={VEL 50.0000,ACC 100.000,APO_DIST 250.000,APO_MODE #CDIS,GEAR_JERK 100.000,EXAX_IGN 0}

DECL E6POS XP330={X 2286.18115,Y 0.000230411548,Z 1849.57446,A -179.999893,B 66.9998779,C -179.999878,S 2,T 35,E1 0.0,E2 0.0,E3 0.0,E4 0.0,E5 0.0,E6 0.0}
DECL FDAT FP330={TOOL_NO 1,BASE_NO 0,IPO_FRAME #BASE,POINT2[] " "}
DECL PDAT PPDAT30={VEL 50.0000,ACC 100.000,APO_DIST 250.000,APO_MODE #CDIS,GEAR_JERK 100.000,EXAX_IGN 0}

DECL E6POS XP340={X 2286.18115,Y 0.000230411548,Z 1849.57446,A -179.999893,B 66.9998779,C -179.999878,S 2,T 35,E1 0.0,E2 0.0,E3 0.0,E4 0.0,E5 0.0,E6 0.0}
DECL FDAT FP340={TOOL_NO 1,BASE_NO 0,IPO_FRAME #BASE,POINT2[] " "}
DECL PDAT PPDAT31={VEL 50.0000,ACC 100.000,APO_DIST 250.000,APO_MODE #CDIS,GEAR_JERK 100.000,EXAX_IGN 0}

DECL E6POS XP350={X 2286.18115,Y 0.000230411548,Z 1849.57446,A -179.999893,B 66.9998779,C -179.999878,S 2,T 35,E1 0.0,E2 0.0,E3 0.0,E4 0.0,E5 0.0,E6 0.0}
DECL FDAT FP350={TOOL_NO 1,BASE_NO 0,IPO_FRAME #BASE,POINT2[] " "}
DECL LDAT LCPDAT13={VEL 0.500000,ACC 100.000,APO_DIST 500.000,APO_FAC 50.0000,AXIS_VEL 100.000,AXIS_ACC 100.000,ORI_TYP #VAR,CIRC_TYP #BASE,JERK_FAC 50.0000,GEAR_JERK 100.000,EXAX_IGN 0,CB {AUX_PT {ORI #CONSIDER,E1 #CONSIDER,E2 #CONSIDER,E3 #CONSIDER,E4 #CONSIDER,E5 #CONSIDER,E6 #CONSIDER},TARGET_PT {ORI #INTERPOLATE,E1 #INTERPOLATE,E2 #INTERPOLATE,E3 #INTERPOLATE,E4 #INTERPOLATE,E5 #INTERPOLATE,E6 #INTERPOLATE}}}
DECL LDAT LCPDAT14={VEL 0.500000,ACC 100.000,APO_DIST 500.000,APO_FAC 50.0000,AXIS_VEL 100.000,AXIS_ACC 100.000,ORI_TYP #VAR,CIRC_TYP #BASE,JERK_FAC 50.0000,GEAR_JERK 100.000,EXAX_IGN 0,CB {AUX_PT {ORI #CONSIDER,E1 #CONSIDER,E2 #CONSIDER,E3 #CONSIDER,E4 #CONSIDER,E5 #CONSIDER,E6 #CONSIDER},TARGET_PT {ORI #INTERPOLATE,E1 #INTERPOLATE,E2 #INTERPOLATE,E3 #INTERPOLATE,E4 #INTERPOLATE,E5 #INTERPOLATE,E6 #INTERPOLATE}}}
DECL PDAT PPDAT32={VEL 50.0000,ACC 100.000,APO_DIST 250.000,APO_MODE #CDIS,GEAR_JERK 100.000,EXAX_IGN 0}
DECL PDAT PPDAT33={VEL 50.0000,ACC 100.000,APO_DIST 250.000,APO_MODE #CDIS,GEAR_JERK 100.000,EXAX_IGN 0}
DECL PDAT PPDAT34={VEL 50.0000,ACC 100.000,APO_DIST 250.000,APO_MODE #CDIS,GEAR_JERK 100.000,EXAX_IGN 0}
DECL PDAT PPDAT35={VEL 50.0000,ACC 100.000,APO_DIST 250.000,APO_MODE #CDIS,GEAR_JERK 100.000,EXAX_IGN 0}

;***************************************************
;Sprue Deposit Declarations*************************
;***************************************************
DECL E6POS XP400={X 2198.25366,Y -125.542969,Z 1747.09790,A 176.729721,B 44.9991875,C 179.999023,S 2,T 34,E1 0.0,E2 0.0,E3 0.0,E4 0.0,E5 0.0,E6 0.0}
DECL FDAT FP400={TOOL_NO 1,BASE_NO 0,IPO_FRAME #BASE,POINT2[] " "}
DECL PDAT PPDAT36={VEL 100.000,ACC 100.000,APO_DIST 500.000,APO_MODE #CDIS,GEAR_JERK 100.000,EXAX_IGN 0}

DECL E6POS XP410={X 2390.31812,Y -1925.40979,Z 1762.14600,A 95.1891937,B -41.9596901,C 111.171272,S 2,T 42,E1 0.0,E2 0.0,E3 0.0,E4 0.0,E5 0.0,E6 0.0}
DECL FDAT FP410={TOOL_NO 1,BASE_NO 0,IPO_FRAME #BASE,POINT2[] " "}
DECL PDAT PPDAT37={VEL 100.000,ACC 100.000,APO_DIST 500.000,APO_MODE #CDIS,GEAR_JERK 100.000,EXAX_IGN 0}

DECL E6POS XP420={X 2979.03320,Y 1211.17944,Z 1330.26062,A 178.656723,B 30.7819328,C 173.526840,S 2,T 35,E1 0.0,E2 0.0,E3 0.0,E4 0.0,E5 0.0,E6 0.0}
DECL FDAT FP420={TOOL_NO 1,BASE_NO 0,IPO_FRAME #BASE,POINT2[] " "}
DECL PDAT PPDAT38={VEL 100.000,ACC 100.000,APO_DIST 500.000,APO_MODE #CDIS,GEAR_JERK 100.000,EXAX_IGN 0}

DECL E6POS XP430={X 2984.07520,Y 1239.72351,Z 1312.65625,A 178.739960,B 30.1429787,C 173.743881,S 2,T 35,E1 0.0,E2 0.0,E3 0.0,E4 0.0,E5 0.0,E6 0.0}
DECL FDAT FP430={TOOL_NO 1,BASE_NO 0,IPO_FRAME #BASE,POINT2[] " "}
DECL PDAT PPDAT39={VEL 100.000,ACC 100.000,APO_DIST 250.000,APO_MODE #CDIS,GEAR_JERK 100.000,EXAX_IGN 0}

DECL E6POS XP440={X 2987.33838,Y 1828.17041,Z 899.984924,A -179.999908,B 18.3625202,C -179.999237,S 2,T 35,E1 0.0,E2 0.0,E3 0.0,E4 0.0,E5 0.0,E6 0.0}
DECL FDAT FP440={TOOL_NO 1,BASE_NO 0,IPO_FRAME #BASE,POINT2[] " "}
DECL PDAT PPDAT40={VEL 100.000,ACC 100.000,APO_DIST 250.000,APO_MODE #CDIS,GEAR_JERK 100.000,EXAX_IGN 0}

DECL E6POS XP450={X 3200.05078,Y -2259.43604,Z 372.462280,A 0.167516440,B -65.0715408,C -179.711563,S 2,T 42,E1 0.0,E2 0.0,E3 0.0,E4 0.0,E5 0.0,E6 0.0}
DECL FDAT FP450={TOOL_NO 1,BASE_NO 0,IPO_FRAME #BASE,POINT2[] " "}
DECL LDAT LCPDAT15={VEL 1.00000,ACC 100.000,APO_DIST 500.000,APO_FAC 50.0000,AXIS_VEL 100.000,AXIS_ACC 100.000,ORI_TYP #VAR,CIRC_TYP #BASE,JERK_FAC 50.0000,GEAR_JERK 100.000,EXAX_IGN 0,CB {AUX_PT {ORI #CONSIDER,E1 #CONSIDER,E2 #CONSIDER,E3 #CONSIDER,E4 #CONSIDER,E5 #CONSIDER,E6 #CONSIDER},TARGET_PT {ORI #INTERPOLATE,E1 #INTERPOLATE,E2 #INTERPOLATE,E3 #INTERPOLATE,E4 #INTERPOLATE,E5 #INTERPOLATE,E6 #INTERPOLATE}}}
DECL LDAT LCPDAT16={VEL 1.00000,ACC 100.000,APO_DIST 500.000,APO_FAC 50.0000,AXIS_VEL 100.000,AXIS_ACC 100.000,ORI_TYP #VAR,CIRC_TYP #BASE,JERK_FAC 50.0000,GEAR_JERK 100.000,EXAX_IGN 0,CB {AUX_PT {ORI #CONSIDER,E1 #CONSIDER,E2 #CONSIDER,E3 #CONSIDER,E4 #CONSIDER,E5 #CONSIDER,E6 #CONSIDER},TARGET_PT {ORI #INTERPOLATE,E1 #INTERPOLATE,E2 #INTERPOLATE,E3 #INTERPOLATE,E4 #INTERPOLATE,E5 #INTERPOLATE,E6 #INTERPOLATE}}}
DECL PDAT PPDAT41={VEL 100.000,ACC 100.000,APO_DIST 250.000,APO_MODE #CDIS,GEAR_JERK 100.000,EXAX_IGN 0}
DECL PDAT PPDAT42={VEL 100.000,ACC 100.000,APO_DIST 250.000,APO_MODE #CDIS,GEAR_JERK 100.000,EXAX_IGN 0}
DECL PDAT PPDAT43={VEL 100.000,ACC 100.000,APO_DIST 250.000,APO_MODE #CDIS,GEAR_JERK 100.000,EXAX_IGN 0}
DECL PDAT PPDAT44={VEL 100.000,ACC 100.000,APO_DIST 250.000,APO_MODE #CDIS,GEAR_JERK 100.000,EXAX_IGN 0}
DECL E6POS XP460={X 2893.71240,Y -2080.63940,Z 947.761169,A 10.9759569,B -62.9248276,C 168.505783,S 2,T 42,E1 0.0,E2 0.0,E3 0.0,E4 0.0,E5 0.0,E6 0.0}
DECL FDAT FP460={TOOL_NO 1,BASE_NO 0,IPO_FRAME #BASE,POINT2[] " "}
DECL PDAT PPDAT79={VEL 100.000,ACC 100.000,APO_DIST 500.000,APO_MODE #CDIS,GEAR_JERK 100.000,EXAX_IGN 0}
DECL E6POS XP470={X 1514.31299,Y -2306.02930,Z 1013.68066,A 179.385300,B 39.6570168,C -179.717957,S 2,T 10,E1 0.0,E2 0.0,E3 0.0,E4 0.0,E5 0.0,E6 0.0}
DECL FDAT FP470={TOOL_NO 1,BASE_NO 0,IPO_FRAME #BASE,POINT2[] " "}
DECL PDAT PPDAT80={VEL 100.000,ACC 100.000,APO_DIST 500.000,APO_MODE #CDIS,GEAR_JERK 100.000,EXAX_IGN 0}

;***************************************************
;Turning station Declarations***********************
;***************************************************
DECL E6POS XP600={X 1359.73181,Y -2243.16748,Z 519.965149,A 179.272369,B 79.2788925,C 178.900391,S 2,T 10,E1 0.0,E2 0.0,E3 0.0,E4 0.0,E5 0.0,E6 0.0}
DECL FDAT FP600={TOOL_NO 1,BASE_NO 0,IPO_FRAME #BASE,POINT2[] " "}
DECL PDAT PPDAT45={VEL 100.000,ACC 100.000,APO_DIST 250.000,APO_MODE #CDIS,GEAR_JERK 100.000,EXAX_IGN 0}

DECL E6POS XP610={X 912.978516,Y -2267.28638,Z -268.156,A 179.234726,B 79.2788925,C 178.900421,S 2,T 10,E1 0.0,E2 0.0,E3 0.0,E4 0.0,E5 0.0,E6 0.0}
DECL FDAT FP610={TOOL_NO 1,BASE_NO 0,IPO_FRAME #BASE,POINT2[] " "}
DECL PDAT PPDAT46={VEL 100.000,ACC 100.000,APO_DIST 250.000,APO_MODE #CDIS,GEAR_JERK 100.000,EXAX_IGN 0}

DECL E6POS XP620={X 912.978638,Y -2269.34033,Z -913.837036,A 179.234726,B 79.2788925,C 178.900421,S 2,T 10,E1 0.0,E2 0.0,E3 0.0,E4 0.0,E5 0.0,E6 0.0}
DECL FDAT FP620={TOOL_NO 1,BASE_NO 0,IPO_FRAME #BASE,POINT2[] " "}
DECL PDAT PPDAT47={VEL 100.000,ACC 100.000,APO_DIST 250.000,APO_MODE #CDIS,GEAR_JERK 100.000,EXAX_IGN 0}

DECL E6POS XP630={X 1634.41479,Y -2205.25439,Z -1087.55615,A 0.288036913,B 56.0250549,C -0.0289533697,S 2,T 8,E1 0.0,E2 0.0,E3 0.0,E4 0.0,E5 0.0,E6 0.0}
DECL FDAT FP630={TOOL_NO 1,BASE_NO 0,IPO_FRAME #BASE,POINT2[] " "}
DECL PDAT PPDAT48={VEL 100.000,ACC 100.000,APO_DIST 250.000,APO_MODE #CDIS,GEAR_JERK 100.000,EXAX_IGN 0}

DECL E6POS XP640={X 2064.59863,Y -2248.80420,Z -849.299133,A 0.255158484,B 52.3243294,C -0.0588298254,S 2,T 10,E1 0.0,E2 0.0,E3 0.0,E4 0.0,E5 0.0,E6 0.0}
DECL FDAT FP640={TOOL_NO 1,BASE_NO 0,IPO_FRAME #BASE,POINT2[] " "}
DECL PDAT PPDAT49={VEL 100.000,ACC 100.000,APO_DIST 250.000,APO_MODE #CDIS,GEAR_JERK 100.000,EXAX_IGN 0}

DECL E6POS XP650={X 2147.17285,Y -2252.73975,Z -631.487671,A 0.240884677,B 49.6522102,C -0.0771938488,S 2,T 10,E1 0.0,E2 0.0,E3 0.0,E4 0.0,E5 0.0,E6 0.0}
DECL FDAT FP650={TOOL_NO 1,BASE_NO 0,IPO_FRAME #BASE,POINT2[] " "}
DECL LDAT LCPDAT17={VEL 0.500000,ACC 100.000,APO_DIST 500.000,APO_FAC 50.0000,AXIS_VEL 100.000,AXIS_ACC 100.000,ORI_TYP #VAR,CIRC_TYP #BASE,JERK_FAC 50.0000,GEAR_JERK 100.000,EXAX_IGN 0,CB {AUX_PT {ORI #CONSIDER,E1 #CONSIDER,E2 #CONSIDER,E3 #CONSIDER,E4 #CONSIDER,E5 #CONSIDER,E6 #CONSIDER},TARGET_PT {ORI #INTERPOLATE,E1 #INTERPOLATE,E2 #INTERPOLATE,E3 #INTERPOLATE,E4 #INTERPOLATE,E5 #INTERPOLATE,E6 #INTERPOLATE}}}
DECL LDAT LCPDAT18={VEL 0.500000,ACC 100.000,APO_DIST 500.000,APO_FAC 50.0000,AXIS_VEL 100.000,AXIS_ACC 100.000,ORI_TYP #VAR,CIRC_TYP #BASE,JERK_FAC 50.0000,GEAR_JERK 100.000,EXAX_IGN 0,CB {AUX_PT {ORI #CONSIDER,E1 #CONSIDER,E2 #CONSIDER,E3 #CONSIDER,E4 #CONSIDER,E5 #CONSIDER,E6 #CONSIDER},TARGET_PT {ORI #INTERPOLATE,E1 #INTERPOLATE,E2 #INTERPOLATE,E3 #INTERPOLATE,E4 #INTERPOLATE,E5 #INTERPOLATE,E6 #INTERPOLATE}}}
DECL PDAT PPDAT51={VEL 100.000,ACC 100.000,APO_DIST 250.000,APO_MODE #CDIS,GEAR_JERK 100.000,EXAX_IGN 0}
DECL PDAT PPDAT52={VEL 100.000,ACC 100.000,APO_DIST 250.000,APO_MODE #CDIS,GEAR_JERK 100.000,EXAX_IGN 0}
DECL PDAT PPDAT53={VEL 100.000,ACC 100.000,APO_DIST 250.000,APO_MODE #CDIS,GEAR_JERK 100.000,EXAX_IGN 0}
DECL PDAT PPDAT54={VEL 100.000,ACC 100.000,APO_DIST 250.000,APO_MODE #CDIS,GEAR_JERK 100.000,EXAX_IGN 0}

DECL PDAT PPDAT81={VEL 100.000,ACC 100.000,APO_DIST 500.000,APO_MODE #CDIS,GEAR_JERK 100.000,EXAX_IGN 0}
DECL FDAT FP660={TOOL_NO 1,BASE_NO 0,IPO_FRAME #BASE,POINT2[] " "}
DECL E6POS XP660={X 2045.59509,Y -2216.04639,Z 722.229797,A -178.599548,B 50.4192886,C -178.898575,S 2,T 10,E1 0.0,E2 0.0,E3 0.0,E4 0.0,E5 0.0,E6 0.0}
DECL LDAT LCPDAT26={VEL 2.00000,ACC 100.000,APO_DIST 500.000,APO_FAC 50.0000,AXIS_VEL 100.000,AXIS_ACC 100.000,ORI_TYP #VAR,CIRC_TYP #BASE,JERK_FAC 50.0000,GEAR_JERK 100.000,EXAX_IGN 0,CB {AUX_PT {ORI #CONSIDER,E1 #CONSIDER,E2 #CONSIDER,E3 #CONSIDER,E4 #CONSIDER,E5 #CONSIDER,E6 #CONSIDER},TARGET_PT {ORI #INTERPOLATE,E1 #INTERPOLATE,E2 #INTERPOLATE,E3 #INTERPOLATE,E4 #INTERPOLATE,E5 #INTERPOLATE,E6 #INTERPOLATE}}}
DECL FDAT FP670={TOOL_NO 1,BASE_NO 0,IPO_FRAME #BASE,POINT2[] " "}
DECL E6POS XP670={X 2045.59509,Y -2264.11572,Z 541.635559,A -176.950058,B 50.3662491,C -176.757690,S 2,T 10,E1 0.0,E2 0.0,E3 0.0,E4 0.0,E5 0.0,E6 0.0}

;***************************************************
;RFID Declarations**********************************
;***************************************************
DECL E6POS XP800={X 1097.71228,Y -2424.92725,Z 738.086670,A 170.962936,B 43.0366020,C -179.002792,S 2,T 10,E1 0.0,E2 0.0,E3 0.0,E4 0.0,E5 0.0,E6 0.0}
DECL FDAT FP800={TOOL_NO 1,BASE_NO 0,IPO_FRAME #BASE,POINT2[] " "}
DECL PDAT PPDAT55={VEL 100.000,ACC 100.000,APO_DIST 250.000,APO_MODE #CDIS,GEAR_JERK 100.000,EXAX_IGN 0}

DECL E6POS XP810={X 1050.91321,Y -2472.18701,Z 296.073547,A 0.474112332,B 59.2422791,C 119.543030,S 2,T 10,E1 0.0,E2 0.0,E3 0.0,E4 0.0,E5 0.0,E6 0.0}
DECL FDAT FP810={TOOL_NO 1,BASE_NO 0,IPO_FRAME #BASE,POINT2[] " "}
DECL PDAT PPDAT56={VEL 100.000,ACC 100.000,APO_DIST 250.000,APO_MODE #CDIS,GEAR_JERK 100.000,EXAX_IGN 0}

DECL E6POS XP820={X 1034.56946,Y -2618.79224,Z -1467.73376,A -0.0106553063,B 45.0740700,C -179.986282,S 2,T 8,E1 0.0,E2 0.0,E3 0.0,E4 0.0,E5 0.0,E6 0.0}
DECL FDAT FP820={TOOL_NO 1,BASE_NO 0,IPO_FRAME #BASE,POINT2[] " "}
DECL PDAT PPDAT57={VEL 100.000,ACC 100.000,APO_DIST 250.000,APO_MODE #CDIS,GEAR_JERK 100.000,EXAX_IGN 0}

DECL E6POS XP840={X 2286.18115,Y 0.000230411548,Z 1849.57446,A -179.999893,B 66.9998779,C -179.999878,S 2,T 35,E1 0.0,E2 0.0,E3 0.0,E4 0.0,E5 0.0,E6 0.0}
DECL FDAT FP840={TOOL_NO 1,BASE_NO 0,IPO_FRAME #BASE,POINT2[] " "}
DECL PDAT PPDAT58={VEL 100.000,ACC 100.000,APO_DIST 250.000,APO_MODE #CDIS,GEAR_JERK 100.000,EXAX_IGN 0}

DECL E6POS XP830={X 1034.56946,Y -2618.79224,Z -1656.55054,A -0.0106553072,B 45.0740700,C -179.986282,S 2,T 8,E1 0.0,E2 0.0,E3 0.0,E4 0.0,E5 0.0,E6 0.0}
DECL FDAT FP830={TOOL_NO 1,BASE_NO 0,IPO_FRAME #BASE,POINT2[] " "}
DECL PDAT PPDAT59={VEL 100.000,ACC 100.000,APO_DIST 250.000,APO_MODE #CDIS,GEAR_JERK 100.000,EXAX_IGN 0}

DECL E6POS XP850={X 666666.688,Y 66.6000,Z 666.660,A 6.60000,B 66.6600,C 666.600,S 0,T 0,E1 0.0,E2 0.0,E3 0.0,E4 0.0,E5 0.0,E6 0.0}
DECL FDAT FP850={TOOL_NO 1,BASE_NO 0,IPO_FRAME #BASE,POINT2[] " "}
DECL LDAT LCPDAT19={VEL 0.500000,ACC 100.000,APO_DIST 500.000,APO_FAC 50.0000,AXIS_VEL 100.000,AXIS_ACC 100.000,ORI_TYP #VAR,CIRC_TYP #BASE,JERK_FAC 50.0000,GEAR_JERK 100.000,EXAX_IGN 0,CB {AUX_PT {ORI #CONSIDER,E1 #CONSIDER,E2 #CONSIDER,E3 #CONSIDER,E4 #CONSIDER,E5 #CONSIDER,E6 #CONSIDER},TARGET_PT {ORI #INTERPOLATE,E1 #INTERPOLATE,E2 #INTERPOLATE,E3 #INTERPOLATE,E4 #INTERPOLATE,E5 #INTERPOLATE,E6 #INTERPOLATE}}}
DECL LDAT LCPDAT20={VEL 0.500000,ACC 100.000,APO_DIST 500.000,APO_FAC 50.0000,AXIS_VEL 100.000,AXIS_ACC 100.000,ORI_TYP #VAR,CIRC_TYP #BASE,JERK_FAC 50.0000,GEAR_JERK 100.000,EXAX_IGN 0,CB {AUX_PT {ORI #CONSIDER,E1 #CONSIDER,E2 #CONSIDER,E3 #CONSIDER,E4 #CONSIDER,E5 #CONSIDER,E6 #CONSIDER},TARGET_PT {ORI #INTERPOLATE,E1 #INTERPOLATE,E2 #INTERPOLATE,E3 #INTERPOLATE,E4 #INTERPOLATE,E5 #INTERPOLATE,E6 #INTERPOLATE}}}
DECL PDAT PPDAT60={VEL 100.000,ACC 100.000,APO_DIST 250.000,APO_MODE #CDIS,GEAR_JERK 100.000,EXAX_IGN 0}
DECL PDAT PPDAT61={VEL 100.000,ACC 100.000,APO_DIST 250.000,APO_MODE #CDIS,GEAR_JERK 100.000,EXAX_IGN 0}
DECL PDAT PPDAT62={VEL 100.000,ACC 100.000,APO_DIST 250.000,APO_MODE #CDIS,GEAR_JERK 100.000,EXAX_IGN 0}
DECL PDAT PPDAT63={VEL 100.000,ACC 100.000,APO_DIST 250.000,APO_MODE #CDIS,GEAR_JERK 100.000,EXAX_IGN 0}

DECL FDAT FP860={TOOL_NO 1,BASE_NO 0,IPO_FRAME #BASE,POINT2[] " "}
DECL E6POS XP860={X 666666.688,Y 66.6000,Z 666.660,A 6.60000,B 66.6600,C 666.600,S 0,T 0,E1 0.0,E2 0.0,E3 0.0,E4 0.0,E5 0.0,E6 0.0}
DECL PDAT PPDAT83={VEL 100.000,ACC 100.000,APO_DIST 500.000,APO_MODE #CDIS,GEAR_JERK 100.000,EXAX_IGN 0}

;***************************************************
;Flaming Declarations*******************************
;***************************************************
DECL E6POS XP700={X 2286.18115,Y 0.000230411548,Z 1849.57446,A -179.999893,B 66.9998779,C -179.999878,S 2,T 35,E1 0.0,E2 0.0,E3 0.0,E4 0.0,E5 0.0,E6 0.0}
DECL FDAT FP700={TOOL_NO 1,BASE_NO 0,IPO_FRAME #BASE,POINT2[] " "}
DECL PDAT PPDAT64={VEL 100.000,ACC 100.000,APO_DIST 250.000,APO_MODE #CDIS,GEAR_JERK 100.000,EXAX_IGN 0}

DECL E6POS XP710={X 2286.18115,Y 0.000230411548,Z 1849.57446,A -179.999893,B 66.9998779,C -179.999878,S 2,T 35,E1 0.0,E2 0.0,E3 0.0,E4 0.0,E5 0.0,E6 0.0}
DECL FDAT FP710={TOOL_NO 1,BASE_NO 0,IPO_FRAME #BASE,POINT2[] " "}
DECL PDAT PPDAT65={VEL 100.000,ACC 100.000,APO_DIST 250.000,APO_MODE #CDIS,GEAR_JERK 100.000,EXAX_IGN 0}

DECL E6POS XP720={X 2286.18115,Y 0.000230411548,Z 1849.57446,A -179.999893,B 66.9998779,C -179.999878,S 2,T 35,E1 0.0,E2 0.0,E3 0.0,E4 0.0,E5 0.0,E6 0.0}
DECL FDAT FP720={TOOL_NO 1,BASE_NO 0,IPO_FRAME #BASE,POINT2[] " "}
DECL PDAT PPDAT66={VEL 100.000,ACC 100.000,APO_DIST 250.000,APO_MODE #CDIS,GEAR_JERK 100.000,EXAX_IGN 0}

DECL E6POS XP730={X 2286.18115,Y 0.000230411548,Z 1849.57446,A -179.999893,B 66.9998779,C -179.999878,S 2,T 35,E1 0.0,E2 0.0,E3 0.0,E4 0.0,E5 0.0,E6 0.0}
DECL FDAT FP730={TOOL_NO 1,BASE_NO 0,IPO_FRAME #BASE,POINT2[] " "}
DECL PDAT PPDAT67={VEL 100.000,ACC 100.000,APO_DIST 250.000,APO_MODE #CDIS,GEAR_JERK 100.000,EXAX_IGN 0}

DECL E6POS XP740={X 2286.18115,Y 0.000230411548,Z 1849.57446,A -179.999893,B 66.9998779,C -179.999878,S 2,T 35,E1 0.0,E2 0.0,E3 0.0,E4 0.0,E5 0.0,E6 0.0}
DECL FDAT FP740={TOOL_NO 1,BASE_NO 0,IPO_FRAME #BASE,POINT2[] " "}
DECL PDAT PPDAT68={VEL 100.000,ACC 100.000,APO_DIST 250.000,APO_MODE #CDIS,GEAR_JERK 100.000,EXAX_IGN 0}

DECL E6POS XP750={X 2286.18115,Y 0.000230411548,Z 1849.57446,A -179.999893,B 66.9998779,C -179.999878,S 2,T 35,E1 0.0,E2 0.0,E3 0.0,E4 0.0,E5 0.0,E6 0.0}
DECL FDAT FP750={TOOL_NO 1,BASE_NO 0,IPO_FRAME #BASE,POINT2[] " "}
DECL LDAT LCPDAT21={VEL 0.500000,ACC 100.000,APO_DIST 500.000,APO_FAC 50.0000,AXIS_VEL 100.000,AXIS_ACC 100.000,ORI_TYP #VAR,CIRC_TYP #BASE,JERK_FAC 50.0000,GEAR_JERK 100.000,EXAX_IGN 0,CB {AUX_PT {ORI #CONSIDER,E1 #CONSIDER,E2 #CONSIDER,E3 #CONSIDER,E4 #CONSIDER,E5 #CONSIDER,E6 #CONSIDER},TARGET_PT {ORI #INTERPOLATE,E1 #INTERPOLATE,E2 #INTERPOLATE,E3 #INTERPOLATE,E4 #INTERPOLATE,E5 #INTERPOLATE,E6 #INTERPOLATE}}}

DECL E6POS XP755={X 2286.18115,Y 0.000230411548,Z 1849.57446,A -179.999893,B 66.9998779,C -179.999878,S 2,T 35,E1 0.0,E2 0.0,E3 0.0,E4 0.0,E5 0.0,E6 0.0}
DECL FDAT FP755={TOOL_NO 1,BASE_NO 0,IPO_FRAME #BASE,POINT2[] " "}
DECL LDAT LCPDAT22={VEL 0.500000,ACC 100.000,APO_DIST 500.000,APO_FAC 50.0000,AXIS_VEL 100.000,AXIS_ACC 100.000,ORI_TYP #VAR,CIRC_TYP #BASE,JERK_FAC 50.0000,GEAR_JERK 100.000,EXAX_IGN 0,CB {AUX_PT {ORI #CONSIDER,E1 #CONSIDER,E2 #CONSIDER,E3 #CONSIDER,E4 #CONSIDER,E5 #CONSIDER,E6 #CONSIDER},TARGET_PT {ORI #INTERPOLATE,E1 #INTERPOLATE,E2 #INTERPOLATE,E3 #INTERPOLATE,E4 #INTERPOLATE,E5 #INTERPOLATE,E6 #INTERPOLATE}}}

DECL E6POS XP760={X 2286.18115,Y 0.000230411548,Z 1849.57446,A -179.999893,B 66.9998779,C -179.999878,S 2,T 35,E1 0.0,E2 0.0,E3 0.0,E4 0.0,E5 0.0,E6 0.0}
DECL FDAT FP760={TOOL_NO 1,BASE_NO 0,IPO_FRAME #BASE,POINT2[] " "}
DECL LDAT LCPDAT23={VEL 0.500000,ACC 100.000,APO_DIST 500.000,APO_FAC 50.0000,AXIS_VEL 100.000,AXIS_ACC 100.000,ORI_TYP #VAR,CIRC_TYP #BASE,JERK_FAC 50.0000,GEAR_JERK 100.000,EXAX_IGN 0,CB {AUX_PT {ORI #CONSIDER,E1 #CONSIDER,E2 #CONSIDER,E3 #CONSIDER,E4 #CONSIDER,E5 #CONSIDER,E6 #CONSIDER},TARGET_PT {ORI #INTERPOLATE,E1 #INTERPOLATE,E2 #INTERPOLATE,E3 #INTERPOLATE,E4 #INTERPOLATE,E5 #INTERPOLATE,E6 #INTERPOLATE}}}

DECL E6POS XP765={X 2286.18115,Y 0.000230411548,Z 1849.57446,A -179.999893,B 66.9998779,C -179.999878,S 2,T 35,E1 0.0,E2 0.0,E3 0.0,E4 0.0,E5 0.0,E6 0.0}
DECL FDAT FP765={TOOL_NO 1,BASE_NO 0,IPO_FRAME #BASE,POINT2[] " "}
DECL LDAT LCPDAT24={VEL 0.500000,ACC 100.000,APO_DIST 500.000,APO_FAC 50.0000,AXIS_VEL 100.000,AXIS_ACC 100.000,ORI_TYP #VAR,CIRC_TYP #BASE,JERK_FAC 50.0000,GEAR_JERK 100.000,EXAX_IGN 0,CB {AUX_PT {ORI #CONSIDER,E1 #CONSIDER,E2 #CONSIDER,E3 #CONSIDER,E4 #CONSIDER,E5 #CONSIDER,E6 #CONSIDER},TARGET_PT {ORI #INTERPOLATE,E1 #INTERPOLATE,E2 #INTERPOLATE,E3 #INTERPOLATE,E4 #INTERPOLATE,E5 #INTERPOLATE,E6 #INTERPOLATE}}}

DECL E6POS XP770={X 2286.18115,Y 0.000230411548,Z 1849.57446,A -179.999893,B 66.9998779,C -179.999878,S 2,T 35,E1 0.0,E2 0.0,E3 0.0,E4 0.0,E5 0.0,E6 0.0}
DECL FDAT FP770={TOOL_NO 1,BASE_NO 0,IPO_FRAME #BASE,POINT2[] " "}
DECL LDAT LCPDAT25={VEL 0.500000,ACC 100.000,APO_DIST 500.000,APO_FAC 50.0000,AXIS_VEL 100.000,AXIS_ACC 100.000,ORI_TYP #VAR,CIRC_TYP #BASE,JERK_FAC 50.0000,GEAR_JERK 100.000,EXAX_IGN 0,CB {AUX_PT {ORI #CONSIDER,E1 #CONSIDER,E2 #CONSIDER,E3 #CONSIDER,E4 #CONSIDER,E5 #CONSIDER,E6 #CONSIDER},TARGET_PT {ORI #INTERPOLATE,E1 #INTERPOLATE,E2 #INTERPOLATE,E3 #INTERPOLATE,E4 #INTERPOLATE,E5 #INTERPOLATE,E6 #INTERPOLATE}}}
DECL PDAT PPDAT69={VEL 100.000,ACC 100.000,APO_DIST 250.000,APO_MODE #CDIS,GEAR_JERK 100.000,EXAX_IGN 0}
DECL PDAT PPDAT70={VEL 100.000,ACC 100.000,APO_DIST 250.000,APO_MODE #CDIS,GEAR_JERK 100.000,EXAX_IGN 0}
DECL PDAT PPDAT71={VEL 100.000,ACC 100.000,APO_DIST 250.000,APO_MODE #CDIS,GEAR_JERK 100.000,EXAX_IGN 0}
DECL PDAT PPDAT72={VEL 100.000,ACC 100.000,APO_DIST 250.000,APO_MODE #CDIS,GEAR_JERK 100.000,EXAX_IGN 0}

;***************************************************
;******* Declarations without burner ***************
;***************************************************

DECL E6POS XP1000={X 2286.18115,Y 0.000230411548,Z 1849.57446,A -179.999893,B 66.9998779,C -179.999878,S 2,T 35,E1 0.0,E2 0.0,E3 0.0,E4 0.0,E5 0.0,E6 0.0}
DECL FDAT FP1000={TOOL_NO 1,BASE_NO 0,IPO_FRAME #BASE,POINT2[] " "}
DECL PDAT PPDAT73={VEL 100.000,ACC 100.000,APO_DIST 250.000,APO_MODE #CDIS,GEAR_JERK 100.000,EXAX_IGN 0}

DECL E6POS XP1010={X 2286.18115,Y 0.000230411548,Z 1849.57446,A -179.999893,B 66.9998779,C -179.999878,S 2,T 35,E1 0.0,E2 0.0,E3 0.0,E4 0.0,E5 0.0,E6 0.0}
DECL FDAT FP1010={TOOL_NO 1,BASE_NO 0,IPO_FRAME #BASE,POINT2[] " "}
DECL PDAT PPDAT74={VEL 100.000,ACC 100.000,APO_DIST 250.000,APO_MODE #CDIS,GEAR_JERK 100.000,EXAX_IGN 0}

DECL E6POS XP1020={X 2286.18115,Y 0.000230411548,Z 1849.57446,A -179.999893,B 66.9998779,C -179.999878,S 2,T 35,E1 0.0,E2 0.0,E3 0.0,E4 0.0,E5 0.0,E6 0.0}
DECL FDAT FP1020={TOOL_NO 1,BASE_NO 0,IPO_FRAME #BASE,POINT2[] " "}
DECL PDAT PPDAT75={VEL 100.000,ACC 100.000,APO_DIST 250.000,APO_MODE #CDIS,GEAR_JERK 100.000,EXAX_IGN 0}

;***************************************************
;************* Declarations without RFID ***********
;***************************************************

DECL E6POS XP2000={X 1097.71216,Y -2424.92725,Z 738.086853,A 170.962936,B 43.0366058,C -179.002792,S 2,T 10,E1 0.0,E2 0.0,E3 0.0,E4 0.0,E5 0.0,E6 0.0}
DECL FDAT FP2000={TOOL_NO 1,BASE_NO 0,IPO_FRAME #BASE,POINT2[] " "}
DECL PDAT PPDAT76={VEL 100.000,ACC 100.000,APO_DIST 250.000,APO_MODE #CDIS,GEAR_JERK 100.000,EXAX_IGN 0}

DECL E6POS XP2010={X 1050.91321,Y -2472.18701,Z 296.073547,A 0.474112332,B 59.2422791,C 119.543030,S 2,T 10,E1 0.0,E2 0.0,E3 0.0,E4 0.0,E5 0.0,E6 0.0}
DECL FDAT FP2010={TOOL_NO 1,BASE_NO 0,IPO_FRAME #BASE,POINT2[] " "}
DECL PDAT PPDAT77={VEL 100.000,ACC 100.000,APO_DIST 250.000,APO_MODE #CDIS,GEAR_JERK 100.000,EXAX_IGN 0}

DECL E6POS XP2020={X 1050.86816,Y -2439.00195,Z -283.510071,A 6.61404,B 49.1595764,C 154.663208,S 2,T 10,E1 0.0,E2 0.0,E3 0.0,E4 0.0,E5 0.0,E6 0.0}
DECL FDAT FP2020={TOOL_NO 1,BASE_NO 0,IPO_FRAME #BASE,POINT2[] " "}
DECL PDAT PPDAT78={VEL 100.000,ACC 100.000,APO_DIST 250.000,APO_MODE #CDIS,GEAR_JERK 100.000,EXAX_IGN 0}

DECL PDAT PPDAT12={VEL 100.000,ACC 100.000,APO_DIST 500.000,APO_MODE #CDIS,GEAR_JERK 100.000,EXAX_IGN 0}
DECL MODULEPARAM_T LAST_TP_PARAMS={PARAMS[] "Kuka.VelocityFieldEnabled=True; Kuka.ColDetectFieldEnabled=True; Kuka.MovementParameterFieldEnabled=True; Kuka.IsAngleEnabled=False; Kuka.PointName=P20; Kuka.FrameData.base_no=0; Kuka.FrameData.tool_no=1; Kuka.FrameData.ipo_frame=#BASE; Kuka.FrameData.point2=; Kuka.isglobalpoint=False; Kuka.MoveDataPtpName=PDAT2; Kuka.MovementDataPdat.apo_mode=#CDIS; Kuka.MovementDataPdat.apo_dist=250; Kuka.MovementData.vel=100; Kuka.MovementData.acc=100; Kuka.MovementData.exax_ign=0; Kuka.VelocityPtp=100; Kuka.BlendingEnabled=False; Kuka.APXEnabled=False; Kuka.CurrentCDSetIndex=0; Kuka.MoveDataName=CPDAT2; Kuka.MovementData.cb={AUX_PT {ORI #CONSIDER,E1 #CONSIDER,E2 #CONSIDER,E3 #CONSIDER,E4 #CONSIDER,E5 #CONSIDER,E6 #CONSIDER},TARGET_PT {ORI #INTERPOLATE,E1 #INTERPOLATE,E2 #INTERPOLATE,E3 #INTERPOLATE,E4 #INTERPOLATE,E5 #INTERPOLATE,E6 #INTERPOLATE}}; Kuka.MovementData.apo_fac=50; Kuka.MovementData.apo_dist=150; Kuka.MovementData.axis_acc=100; Kuka.MovementData.axis_vel=100; Kuka.MovementData.circ_typ=#BASE; Kuka.MovementData.jerk_fac=50; Kuka.MovementData.ori_typ=#VAR; Kuka.VelocityPath=2     "}
DECL PDAT PPDAT50={VEL 100.000,ACC 100.000,APO_DIST 500.000,APO_MODE #CDIS,GEAR_JERK 100.000,EXAX_IGN 0}


DECL LDAT LCPDAT27={VEL 2.00000,ACC 100.000,APO_DIST 500.000,APO_FAC 50.0000,AXIS_VEL 100.000,AXIS_ACC 100.000,ORI_TYP #VAR,CIRC_TYP #BASE,JERK_FAC 50.0000,GEAR_JERK 100.000,EXAX_IGN 0,CB {AUX_PT {ORI #CONSIDER,E1 #CONSIDER,E2 #CONSIDER,E3 #CONSIDER,E4 #CONSIDER,E5 #CONSIDER,E6 #CONSIDER},TARGET_PT {ORI #INTERPOLATE,E1 #INTERPOLATE,E2 #INTERPOLATE,E3 #INTERPOLATE,E4 #INTERPOLATE,E5 #INTERPOLATE,E6 #INTERPOLATE}}}
DECL PDAT PPDAT82={VEL 100.000,ACC 100.000,APO_DIST 500.000,APO_MODE #CDIS,GEAR_JERK 100.000,EXAX_IGN 0}
DECL LDAT LCPDAT28={VEL 0.500000,ACC 100.000,APO_DIST 500.000,APO_FAC 50.0000,AXIS_VEL 100.000,AXIS_ACC 100.000,ORI_TYP #VAR,CIRC_TYP #BASE,JERK_FAC 50.0000,GEAR_JERK 100.000,EXAX_IGN 0,CB {AUX_PT {ORI #CONSIDER,E1 #CONSIDER,E2 #CONSIDER,E3 #CONSIDER,E4 #CONSIDER,E5 #CONSIDER,E6 #CONSIDER},TARGET_PT {ORI #INTERPOLATE,E1 #INTERPOLATE,E2 #INTERPOLATE,E3 #INTERPOLATE,E4 #INTERPOLATE,E5 #INTERPOLATE,E6 #INTERPOLATE}}}
DECL LDAT LCPDAT29={VEL 0.500000,ACC 100.000,APO_DIST 500.000,APO_FAC 50.0000,AXIS_VEL 100.000,AXIS_ACC 100.000,ORI_TYP #VAR,CIRC_TYP #BASE,JERK_FAC 50.0000,GEAR_JERK 100.000,EXAX_IGN 0,CB {AUX_PT {ORI #CONSIDER,E1 #CONSIDER,E2 #CONSIDER,E3 #CONSIDER,E4 #CONSIDER,E5 #CONSIDER,E6 #CONSIDER},TARGET_PT {ORI #INTERPOLATE,E1 #INTERPOLATE,E2 #INTERPOLATE,E3 #INTERPOLATE,E4 #INTERPOLATE,E5 #INTERPOLATE,E6 #INTERPOLATE}}}

DECL PDAT PPDAT84={VEL 100.000,ACC 100.000,APO_DIST 500.000,APO_MODE #CDIS,GEAR_JERK 100.000,EXAX_IGN 0}
DECL PDAT PPDAT85={VEL 100.000,ACC 100.000,APO_DIST 500.000,APO_MODE #CDIS,GEAR_JERK 100.000,EXAX_IGN 0}
DECL PDAT PPDAT86={VEL 100.000,ACC 100.000,APO_DIST 500.000,APO_MODE #CDIS,GEAR_JERK 100.000,EXAX_IGN 0}
ENDDAT
